FUNCTION_BLOCK MotorVarSpeed_FB
VAR_INPUT
	Run			:	BOOL;
	Direction	:	BOOL;
	ConstSpeed	:	BOOL;
	Velocity	:	INT;
END_VAR
VAR_OUTPUT
	isRunning	:	BOOL;
	iActualVel	:	INT;
END_VAR
VAR
END_VAR

END_FUNCTION_BLOCK

(* stored: Version 1.1.0.1, ProductVersion 3.1.4024.11
   POU MotorVarSpeed_FB: Id {e9de67a0-f478-4523-bff0-bbe131d76573}, SpecialFunc None *)
